(* CoDeSys 2.3.9.28 project: Aula13_ex.pro *)
(* Libraries: Standard.lib 27.1.09 11:27:38, Util.lib 27.1.09 11:27:38, IecSfc.lib*24.11.08 08:07:15, SysLibTime.lib*27.1.09 11:27:38, SysTaskInfo.lib 24.11.08 08:07:15, SYSLIBCALLBACK.LIB 27.1.09 11:27:38 *)

(* PLC configuration (modules and I/O channels)
CPX-CEC [Root] node -1, in %IB0 out %QB0 {StringParam = 2773,0,0,0,0; ByteParam = 0; ByteParam = 31; ByteParam = 0; ByteParam = 0; ByteParam = 0; ByteParam = 0; ByteParam = 0; ByteParam = 0; ByteParam = 2; ByteParam = 0; ByteParam = 0; ByteParam = 0; ByteParam = 32; ByteParam = 0; ByteParam = 0; ByteParam = 5; ByteParam = 0; ByteParam = 0; ByteParam = 0; ByteParam = 0; ByteParam = 0; ByteParam = 0; ByteParam = 0; ByteParam = 0; ByteParam = 14; ByteParam = 240; ByteParam = 192; ByteParam = 168; ByteParam = 2; ByteParam = 10; ByteParam = 255; ByteParam = 255; ByteParam = 0; ByteParam = 0; ByteParam = 192; ByteParam = 168; ByteParam = 1; ByteParam = 1; ByteParam = 192; ByteParam = 168; ByteParam = 2; ByteParam = 10; ByteParam = 255; ByteParam = 255; ByteParam = 0; ByteParam = 0; ByteParam = 192; ByteParam = 168; ByteParam = 1; ByteParam = 1}
  Hexswitch AT %IB0 [HexSwitch] rotary switch 0 = STOP, 1-15 = RUN
  IOModules [CPX_MASTER] node 0, in %IB4 out %QB0
*)

(* Global variable list: Global_Variables *)
VAR_GLOBAL

	START: BOOL;
	STOP : BOOL;
	S1: BOOL;
	S2: BOOL;
	S3: BOOL;
	S4: BOOL;

	M1: BOOL;
	LP: BOOL;
	C1: BOOL;
	C2: BOOL;

	MEM : BOOL;
	MEM2 : BOOL;
	MEM3: BOOL;
	MEM4: BOOL;
	MEM5: BOOL;

	CONT1 : CTU;
	T1 : TON;

END_VAR

(* POU PLC_PRG, ST *)
PROGRAM PLC_PRG
VAR
END_VAR
T1(IN := S3, PT:= T#1s);
CONT1(CU := S4 AND MEM5, RESET := STOP, PV := 2);

IF START AND NOT MEM AND NOT S4 AND NOT LP THEN
	M1 := TRUE;
	C1 := TRUE;
	C2 := TRUE;
	MEM := TRUE;
END_IF



IF S1 THEN
	C1 := FALSE;
	MEM3 := TRUE;
END_IF



IF S2 AND MEM3 THEN
	M1 := FALSE;
	C2 := FALSE;
	MEM3 := FALSE;
	MEM4 := TRUE;
END_IF



IF T1.Q AND MEM4 THEN
	C2 := TRUE;
	M1 := TRUE;
	MEM4 := FALSE;
	MEM5 := TRUE;
END_IF



IF S4 AND MEM5 THEN
	MEM2 := TRUE;
	MEM5 := FALSE;
	M1 := FALSE;
END_IF



IF NOT S4 AND MEM2 THEN
	C2 := TRUE;
	C1 := TRUE;
	MEM2 := FALSE;
	M1 := TRUE;
END_IF



IF CONT1.Q THEN
	LP := TRUE;
	C1 := FALSE;
	M1 := FALSE;
	MEM2 := FALSE;
	MEM3 := FALSE;
	MEM4 := FALSE;
	MEM5 := FALSE;
END_IF


IF STOP THEN
	LP := FALSE;
	M1 := FALSE;
	C1 := FALSE;
	C2 := TRUE;
	MEM := FALSE;
	MEM2 := FALSE;
	MEM3 := FALSE;
	MEM4 := FALSE;
	MEM5 := FALSE;
END_IF
END_PROGRAM

(* Visualisation screen
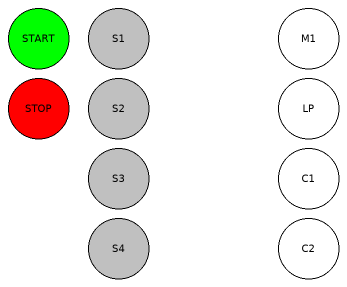
ellipse at (130,50)-(191,111): text "S1"; alarm colour if S1; taps S1
ellipse at (130,120)-(191,181): text "S2"; alarm colour if S2; toggles S2
ellipse at (130,190)-(191,251): text "S3"; alarm colour if S3; toggles S3
ellipse at (130,260)-(191,321): text "S4"; alarm colour if S4; taps S4
ellipse at (50,50)-(111,111): text "START"; alarm colour if START; taps START
ellipse at (50,120)-(111,181): text "STOP"; alarm colour if STOP; taps STOP
ellipse at (320,50)-(381,111): text "M1"; alarm colour if M1
ellipse at (320,120)-(381,181): text "LP"; alarm colour if LP
ellipse at (320,190)-(381,251): text "C1"; alarm colour if C1
ellipse at (320,260)-(381,321): text "C2"; alarm colour if C2
*)
